(* IEC 61131-3 sources: Projecte/smart_office, 5 files *)

(* ---- control_cortines.st ---- *)
// 4. Màquina d'Estats
IF #HabilitarControl THEN
    CASE #Estat OF
        0: // Repòs
            #EnMoviment := FALSE;
            #VelocitatActual := 0.0;
            #RampaActiva := FALSE;
            #ComptePasos := 0;
            IF #sPosicioActual_Passos <> #PosicioDesitjadaPassos THEN
                #Estat := 10; // Passar a Preparar Moviment
            END_IF;

        10: // Preparar Moviment
            #EnMoviment := TRUE;
            #DireccioAssignada := (#PosicioDesitjadaPassos > #sPosicioActual_Passos) XOR NOT #DireccioPerObrir;
            #VelocitatActual := 10.0; // Velocitat inicial
            #RampaActiva := TRUE;
            #ComptePasos := 0;
            #Estat := 20; // Passar a Moviment
            #sTimerPols(IN := TRUE,
                        PT := #PT);
            #PasActual := FALSE;

        20: // Moviment
            #sTimerPols(IN := TRUE,
                        PT := #TempsPolsActual);

            IF #sTimerPols.Q THEN
                // Reiniciar el temporitzador per al següent pols

                // Generar pols i actualitzar direcció
                #PasActual := NOT #PasActual;
                #MotorPols := #PasActual;
                #MotorDireccio := #DireccioAssignada;

                // Actualitzar posició segons la direcció
                IF #DireccioAssignada = #DireccioPerObrir THEN
                    #sPosicioActual_Passos := #sPosicioActual_Passos + 1;
                ELSE
                    #sPosicioActual_Passos := #sPosicioActual_Passos - 1;
                END_IF;

                // Control de Rampa
                IF #RampaActiva THEN
                    #ComptePasos := #ComptePasos + 1;
                    IF #ComptePasos >= #PasosPerRampa THEN
                        #ComptePasos := 0;
                        IF #sPosicioActual_Passos < (#PosicioDesitjadaPassos + #CarreraTotal_Passos / 10) AND
                            #sPosicioActual_Passos > (#PosicioDesitjadaPassos - #CarreraTotal_Passos / 10) THEN
                            // Desaccelerar
                            #VelocitatActual := #VelocitatActual - #Desacceleracio;
                            IF #VelocitatActual <= 10.0 THEN
                                #VelocitatActual := 10.0;
                                #RampaActiva := FALSE; // Fi de la rampa
                            END_IF;
                        ELSE
                            // Accelerar
                            #VelocitatActual := #VelocitatActual + #Acceleracio;
                            IF #VelocitatActual >= 100.0 THEN
                                #VelocitatActual := 100.0;
                            END_IF;
                        END_IF;

                        IF #VelocitatActual <> 0.0 THEN
                            // Conversió més directa i segura
                            #TempsPolsActual := DINT_TO_TIME(REAL_TO_DINT(1000.0 / #VelocitatActual));
                        ELSE
                            #TempsPolsActual := #TempsPolsBase;
                        END_IF;
                    END_IF;
                END_IF;

                // Comprovar posició desitjada (SENSE SENSORS DE LÍMIT)
                IF #sPosicioActual_Passos = #PosicioDesitjadaPassos THEN
                    #Estat := 0; // Aturar moviment
                    #MotorPols := FALSE;
                    #EnMoviment := FALSE;
                    #RampaActiva := FALSE;
                    #ComptePasos := 0;
                END_IF;
            END_IF;

        ELSE // Error
            #Estat := 0;
            #MotorPols := FALSE;
            #EnMoviment := FALSE;
            #RampaActiva := FALSE;
            #ComptePasos := 0;
    END_CASE;
ELSE
    #MotorPols := FALSE;
    #EnMoviment := FALSE;
    #RampaActiva := FALSE;
    #ComptePasos := 0;
END_IF;                // Control de Rampa
                IF #RampaActiva THEN
                    #ComptePasos := #ComptePasos + 1;
                    IF #ComptePasos >= #PasosPerRampa THEN
                        #ComptePasos := 0;
                        IF #sPosicioActual_Passos < (#PosicioDesitjadaPassos + #CarreraTotal_Passos / 10) AND
                            #sPosicioActual_Passos > (#PosicioDesitjadaPassos - #CarreraTotal_Passos / 10) THEN
                            // Desaccelerar
                            #VelocitatActual := #VelocitatActual - #Desacceleracio;
                            IF #VelocitatActual <= 10.0 THEN
                                #VelocitatActual := 10.0;
                                #RampaActiva := FALSE; // Fi de la rampa
                            END_IF;
                        ELSE
                            // Accelerar
                            #VelocitatActual := #VelocitatActual + #Acceleracio;
                            IF #VelocitatActual >= 100.0 THEN
                                #VelocitatActual := 100.0;
                            END_IF;
                        END_IF;

                        IF #VelocitatActual <> 0.0 THEN
                            // Conversió més directa i segura
                            #TempsPolsActual := DINT_TO_TIME(REAL_TO_DINT(1000.0 / #VelocitatActual));
                        ELSE
                            #TempsPolsActual := #TempsPolsBase;
                        END_IF;
                    END_IF;
                END_IF;

                // Comprovar posició desitjada (SENSE SENSORS DE LÍMIT)
                IF #sPosicioActual_Passos = #PosicioDesitjadaPassos THEN
                    #Estat := 0; // Aturar moviment
                    #MotorPols := FALSE;
                    #EnMoviment := FALSE;
                    #RampaActiva := FALSE;
                    #ComptePasos := 0;
                END_IF;
            END_IF;

        ELSE // Error
            #Estat := 0;
            #MotorPols := FALSE;
            #EnMoviment := FALSE;
            #RampaActiva := FALSE;
            #ComptePasos := 0;
    END_CASE;

ELSE
    #MotorPols := FALSE;
    #EnMoviment := FALSE;
    #RampaActiva := FALSE;
    #ComptePasos := 0;
END_IF;

(* ---- control_temperatura.st ---- *)
// BLOC 1: INICIALITZACIÓ I DEFINICIÓ DE VARIABLES
VAR_INPUT
    SetPointNodeRED : Real;  // Setpoint rebut de Node-RED
    sensor_temp_jefe : Int;  // Entrada del sensor de Factory IO (%IW40)
    temperatura_DB : "temperatura_cap_DB";  // Referència al DB de temperatura
END_VAR

VAR_OUTPUT
    TemperaturaNodeRED : Real;  // Temperatura en graus per Node-RED
END_VAR

STATIC
    // Constants del sistema
    TEMP_MIN : Real := 0.0;           // Temperatura mínima permesa (canviat de 15.0)
    TEMP_MAX : Real := 50.0;          // Temperatura màxima permesa (canviat de 30.0)
    ZONA_MORTA : Real := 0.3;         // Marge de zona morta pel control
    HISTERESI : Real := 1.2;          // Factor d'histèresi
    TEMPS_MINIM_CANVI : Time := T#180S; // Temps mínim entre canvis de mode
    TAXA_ESCALFAMENT : Real := 0.1;    // Taxa d'escalfament simulada
    TAXA_REFREDAMENT : Real := 0.05;   // Taxa de refredament simulada

    // Variables de control i estat
    PrimeraExecucio : Bool := TRUE;   // Flag de primera execució
    EstemEnZonaMorta : Bool;          // Control d'histèresi
    ControlActiu : Bool;              // Estat del sistema
    ModeFred : Bool;                  // Mode refrigeració actiu
    ModeCalent : Bool;                // Mode calefacció actiu
    ModeActual : String;              // Mode actual en text

    // Variables de temperatura i sensors
    TemperaturaSimulada : Real;       // Temperatura simulada del sistema
    UltimaTemperaturaReal : Real;     // Última lectura vàlida
    TemperaturaReal : Real;           // Temperatura actual
    TemperaturaEscalada : Real;       // Temperatura processada
    ValorSensor : Real;               // Valor raw del sensor
    Valor_Raw_Sensor : Int;           // Valor enter del sensor

    // Variables de temps i simulació
    TempsActual : Time;               // Temps actual
    TempsAnterior : Time;             // Temps anterior
    DeltaTemps : Real;                // Interval de temps
    ProporcioSimulada : Real;         // Proporció per simulació
    ValorSensorSimulat : Int;         // Valor simulat

    // Variables de sortida i control
    SortidaPID : Real;                // Sortida del controlador PID
    SortidaEscalada : Real;           // Sortida escalada (0-100%)

    // Variables HMI/Monitorització
    HMI_TemperaturaActual : Real;     // Temperatura actual per HMI
    HMI_SetPoint : Real;              // SetPoint actual per HMI
    HMI_ModeActual : String;          // Mode de funcionament per HMI
    HMI_PercentatgeSortida : Real;    // Percentatge sortida per HMI

{REGION 'Declaració de variables PID'}
VAR_INPUT
    EN : Bool;              // Habilitació del PID
    Setpoint : Real;        // Valor desitjat de temperatura
    Input : Real;           // Valor actual de temperatura
END_VAR

VAR_OUTPUT
    Output : Real;          // Sortida del controlador PID
END_VAR

// 1. PROCESSAMENT DEL SENSOR DE TEMPERATURA
// Inicialització de variables de simulació
IF #PrimeraExecucio THEN
    #PrimeraExecucio := FALSE;
    #TemperaturaSimulada := #TEMP_MIN;
    #UltimaTemperaturaReal := #TEMP_MIN;
    #TemperaturaEscalada := #TEMP_MIN;
    #TempsAnterior := T#0MS;
END_IF;

// 2. CONTROL PRINCIPAL ON/OFF
IF NOT #ClimaOn THEN
    // Sistema desactivat - Reset de variables
    #ControlActiu := FALSE;
    #SortidaPID := 0.0;
    #SortidaEscalada := 0.0;
    #ModeFred := FALSE;
    #ModeCalent := FALSE;
    #ModeActual := 'OFF';
    // Mantenim la última temperatura quan està apagat
    #TemperaturaEscalada := #TemperaturaSimulada;
ELSE
    #ControlActiu := TRUE;
END_IF;

// 3. ACTUALITZACIÓ DEL TEMPS I SIMULACIÓ
// Actualitzar temps per la simulació utilitzant TON
#TimerSimulacio(IN := TRUE,
                PT := T#1S);  // Actualitzem cada segon

IF #TimerSimulacio.Q THEN
    #TempsActual := #TimerSimulacio.ET;

    // Calcular delta de temps (en segons)
    IF #TempsAnterior = T#0MS THEN
        #DeltaTemps := 0.1;  // Valor inicial per evitar pics
    ELSE
        #DeltaTemps := DINT_TO_REAL(TIME_TO_DINT(#TempsActual - #TempsAnterior)) / 1000.0;
    END_IF;

    #TempsAnterior := #TempsActual;
    #TimerSimulacio(IN := FALSE,
                    PT := T#1S);  // Reiniciar el timer
END_IF;

// Processar valor del sensor abans de la simulació
#ValorSensor := INT_TO_REAL(#sensor_temp_jefe);
#Valor_Raw_Sensor := #sensor_temp_jefe;

// Normalització i escalat del sensor actual
#Proporcio := #ValorSensor / 27648.0;
#TemperaturaReal := #Proporcio * (#TEMP_MAX - #TEMP_MIN) + #TEMP_MIN;
#TemperaturaEscalada := #TemperaturaReal;  // Utilitzem la temperatura real en lloc de la simulada

// Assignar al DB de temperatura utilitzant la referència
#temperatura_DB.TemperaturaEscalada := #TemperaturaEscalada;

// Validació del SetPoint
IF #SetPointNodeRED < #TEMP_MIN THEN
    #SetPointNodeRED := #TEMP_MIN;
ELSIF #SetPointNodeRED > #TEMP_MAX THEN
    #SetPointNodeRED := #TEMP_MAX;
END_IF;

// Debug dels valors - Actualitzem sempre
#proporcio_debug := #Proporcio;
#temp_real_debug := #TemperaturaReal;
#setpoint_debug := #SetPointNodeRED;
#temp_entrada_pid := #TemperaturaEscalada;
#setpoint_entrada_pid := #SetPointNodeRED;

// Simulació del comportament tèrmic sempre activa
IF #ControlActiu THEN
    IF #ModeFred THEN
        // Mode refrigeració - La sortida del PID refreda
        #TemperaturaSimulada := #TemperaturaSimulada - (#SortidaEscalada * #TAXA_ESCALFAMENT * #DeltaTemps);
    ELSE
        // Mode calefacció - La sortida del PID escalfa
        #TemperaturaSimulada := #TemperaturaSimulada + (#SortidaEscalada * #TAXA_ESCALFAMENT * #DeltaTemps);
    END_IF;

    // Simular pèrdua natural de temperatura
    IF #TemperaturaSimulada > #TEMP_MIN THEN
        #TemperaturaSimulada := #TemperaturaSimulada - (#TAXA_REFREDAMENT * #DeltaTemps);
    END_IF;

    // Limitar la temperatura simulada
    IF #TemperaturaSimulada < #TEMP_MIN THEN
        #TemperaturaSimulada := #TEMP_MIN;
    ELSIF #TemperaturaSimulada > #TEMP_MAX THEN
        #TemperaturaSimulada := #TEMP_MAX;
    END_IF;

    // Actualitzar temperatura escalada amb la simulada
    #TemperaturaEscalada := #TemperaturaSimulada;

    // Convertir temperatura simulada a format sensor (0-27648)
    #ProporcioSimulada := (#TemperaturaSimulada - #TEMP_MIN) / (#TEMP_MAX - #TEMP_MIN);
    #ValorSensorSimulat := REAL_TO_INT(#ProporcioSimulada * 27648.0);

    // Assignar al tag del sensor
    "sensor_temp_jefe" := #ValorSensorSimulat;
END_IF;

// Debug dels valors - Actualitzem sempre
#proporcio_debug := #ProporcioSimulada;
#temp_real_debug := #TemperaturaSimulada;
#setpoint_debug := #SetPointNodeRED;
#temp_entrada_pid := #TemperaturaEscalada;
#setpoint_entrada_pid := #SetPointNodeRED;

// 3. GESTIÓ DE MODES AMB TEMPORITZACIÓ
IF #ControlActiu THEN
    // Control de temps mínim entre canvis
    #TimerCanviMode(IN := #BotoFred OR #BotoCalent,
                    PT := #TEMPS_MINIM_CANVI);

    // Canvi de mode amb temporització
    IF #TimerCanviMode.Q THEN
        IF #BotoFred AND NOT #BotoCalent AND NOT #ModeFred THEN
            // Activació mode fred
            #ModeFred := TRUE;
            #ModeCalent := FALSE;
            #ModeActual := 'Fred';
        ELSIF #BotoCalent AND NOT #BotoFred AND NOT #ModeCalent THEN
            // Activació mode calent
            #ModeFred := FALSE;
            #ModeCalent := TRUE;
            #ModeActual := 'Calent';
        END_IF;
    END_IF;

    // 4. CONTROL PID I SORTIDA
    IF #ClimaOn THEN
        // Configuració del PID
        "Control_temperatura_oficina_cap"(
            EN := #ClimaOn,
            Setpoint := #SetPointNodeRED,
            Input := #TemperaturaEscalada
        );

        // Execució del PID si estem fora de la zona morta
        IF NOT #EstemEnZonaMorta THEN
            #SortidaPID := "Control_temperatura_oficina_cap".Output;
            // Gestió mode fred
            IF #ModeFred THEN
                #SortidaPID := -#SortidaPID;
            END_IF;

            // Limitació de la sortida amb més granularitat
            IF #SortidaPID < 0.0 THEN
                #SortidaEscalada := 0.0;
            ELSIF #SortidaPID > 100.0 THEN
                #SortidaEscalada := 100.0;
            ELSE
                #SortidaEscalada := #SortidaPID;
            END_IF;
        END_IF;
    ELSE
        "Control_temperatura_oficina_cap"(EN := FALSE);
    END_IF;
END_IF;

// BLOC 5: PROCESSAMENT DE SORTIDES
// Convertir temperatura simulada a format sensor
#ProporcioSimulada := (#TemperaturaSimulada - #TEMP_MIN) / (#TEMP_MAX - #TEMP_MIN);
#ValorSensorSimulat := REAL_TO_INT(#ProporcioSimulada * 27648.0);

// Assignar al tag del sensor (simulació)
"sensor_temp_jefe" := #ValorSensorSimulat;

// Actualitzar sortides físiques
#refredament := #ControlActiu AND #ModeFred AND (#SortidaEscalada > 10.0);
#calefaccio := #ControlActiu AND #ModeCalent AND (#SortidaEscalada > 10.0);

// BLOC 6: DIAGNÒSTIC I MONITORITZACIÓ
// Variables per monitorització
#HMI_TemperaturaActual := #TemperaturaSimulada;
#HMI_SetPoint := #SetPointNodeRED;
#HMI_ModeActual := #ModeActual;
#HMI_PercentatgeSortida := #SortidaEscalada;

// Actualitzar temperatura per Node-RED
#Temperatura := #TemperaturaEscalada;

(* ---- control_temperatura_final.st ---- *)
// BLOC 1: INICIALITZACIÓ I DEFINICIÓ DE VARIABLES
VAR_INPUT
    ClimaOn : Bool;         // Interruptor principal del sistema (0.0)
    BotoFred : Bool;        // Botó per activar mode refrigeració (des de Node-RED)
    BotoCalent : Bool;      // Botó per activar mode calefacció (des de Node-RED)
    SetPointNodeRED : Real; // Punt de consigna rebut de Node-RED (2.0)
    sensor_temp_jefe : Int; // Entrada del sensor de Factory IO (%IW40)
END_VAR

VAR_OUTPUT
    refredament : Bool;          // Sortida de refrigeració (276.0)
    calefaccio : Bool;          // Sortida de calefacció (276.1)
    HMI_TemperaturaActual : Real; // Temperatura actual per HMI (278.0)
    HMI_SetPoint : Real;         // Punt de consigna per HMI (282.0)
    HMI_ModeActual : String;     // Mode actual per HMI (286.0)
    HMI_PercentatgeSortida : Real; // Percentatge sortida per HMI (542.0)
    TemperaturaNodeRED : Real;   // Temperatura per Node-RED
END_VAR

STATIC
    // Constants del sistema
    TEMP_MIN : Real := 0.0;            // Temperatura mínima (680.0)
    TEMP_MAX : Real := 50.0;           // Temperatura màxima (684.0)
    ZONA_MORTA : Real := 0.3;          // Marge de zona morta (572.0)
    HISTERESI : Real := 1.2;           // Factor d'histèresi (688.0)
    TEMPS_MINIM_CANVI : Time := T#180S; // Temps mínim entre canvis (568.0)

    // Variables de control i estat
    ControlActiu : Bool;               // Estat del sistema (14.0)
    ModeFred : Bool := FALSE;          // Mode refrigeració actiu (546.0)
    ModeCalent : Bool := FALSE;        // Mode calefacció actiu (546.1)
    ModeActual : String;               // Mode actual (16.0)
    EstemEnZonaMorta : Bool;           // Control d'histèresi (600.0)

    // Variables de temperatura i sensors
    TemperaturaReal : Real;            // Temperatura actual (606.0)
    TemperaturaEscalada : Real;        // Temperatura processada (6.0)
    ValorSensor : Real;                // Valor del sensor (610.0)
    Proporcio : Real;                  // Proporció escalada (548.0)

    // Variables de sortida i control
    SortidaPID : Real;                 // Sortida del controlador PID (10.0)
    SortidaEscalada : Real;            // Sortida escalada 0-100% (272.0)

    // Timer per canvi de mode
    TimerCanviMode : TON_TIME;         // Timer pel canvi de mode (552.0)
END_STATIC

BEGIN
// BLOC 2: PROCESSAMENT DEL SENSOR
// Lectura i processament del sensor
#ValorSensor := INT_TO_REAL(#sensor_temp_jefe);  // Llegim el valor del potenciòmetre
#Proporcio := #ValorSensor / 27648.0;            // Normalitzem a 0-1
#TemperaturaReal := #Proporcio * (#TEMP_MAX - #TEMP_MIN) + #TEMP_MIN;  // Escalem a 0-50°C
#TemperaturaEscalada := #TemperaturaReal;

// BLOC 3: CONTROL PRINCIPAL
IF NOT #ClimaOn THEN
    // Sistema desactivat - Reset de variables
    #ControlActiu := FALSE;
    #SortidaPID := 0.0;
    #SortidaEscalada := 0.0;
    #ModeFred := FALSE;
    #ModeCalent := FALSE;
    #ModeActual := 'Aturat';
ELSE
    #ControlActiu := TRUE;
END_IF;

// BLOC 4: GESTIÓ DE MODES
IF #ControlActiu THEN
    // Control de temps mínim entre canvis
    #TimerCanviMode(IN := (#BotoFred AND NOT #ModeFred) OR (#BotoCalent AND NOT #ModeCalent),
                    PT := #TEMPS_MINIM_CANVI);

    // Actualització de modes amb temporització
    IF #TimerCanviMode.Q THEN
        #ModeFred := #BotoFred AND NOT #BotoCalent;
        #ModeCalent := #BotoCalent AND NOT #BotoFred;

        IF #ModeFred THEN
            #ModeActual := 'Fred';
        ELSIF #ModeCalent THEN
            #ModeActual := 'Calent';
        ELSE
            #ModeActual := 'Aturat';
        END_IF;
    END_IF;

    // BLOC 5: CONTROL PID
    IF #ClimaOn THEN
        // PID Mode Fred
        "Control_temperatura_fred"(
            EN := #ControlActiu AND #ModeFred,  // Cambiado de BotoFred a ModeFred
            ManualEnable := FALSE,
            Reset := FALSE,
            Setpoint := #SetPointNodeRED,
            Input := #TemperaturaEscalada,
            ManualValue := 0.0
        );

        // PID Mode Calent
        "Control_temperatura_calent"(
            EN := #ControlActiu AND #ModeCalent,  // Cambiado de BotoCalent a ModeCalent
            ManualEnable := FALSE,
            Reset := FALSE,
            Setpoint := #SetPointNodeRED,
            Input := #TemperaturaEscalada,
            ManualValue := 0.0
        );

        // Actualitzar zona morta
        #EstemEnZonaMorta := ABS(#SetPointNodeRED - #TemperaturaEscalada) < #ZONA_MORTA;

        // Selecció de la sortida segons el mode actiu
        IF #ModeFred AND NOT #EstemEnZonaMorta THEN  // Cambiado de BotoFred a ModeFred
            #SortidaPID := "Control_temperatura_fred".Output;
        ELSIF #ModeCalent AND NOT #EstemEnZonaMorta THEN  // Cambiado de BotoCalent a ModeCalent
            #SortidaPID := "Control_temperatura_calent".Output;
        END_IF;

        // Limitació de la sortida (comuna per ambdós modes)
        IF #SortidaPID < 0.0 THEN
            #SortidaEscalada := 0.0;
        ELSIF #SortidaPID > 100.0 THEN
            #SortidaEscalada := 100.0;
        ELSE
            #SortidaEscalada := #SortidaPID;
        END_IF;
    ELSE
        // Desactivem ambdós PIDs i els posem en mode manual
        "Control_temperatura_fred"(
            EN := FALSE,
            ManualEnable := TRUE,
            Reset := TRUE,
            Setpoint := 0.0,
            Input := 0.0,
            ManualValue := 0.0
        );

        "Control_temperatura_calent"(
            EN := FALSE,
            ManualEnable := TRUE,
            Reset := TRUE,
            Setpoint := 0.0,
            Input := 0.0,
            ManualValue := 0.0
        );
    END_IF;
END_IF;

// BLOC 6: ACTUALITZACIÓ DE SORTIDES
#refredament := #ControlActiu AND #ModeFred;  // En simulació, activem directament amb el mode
#calefaccio := #ControlActiu AND #ModeCalent;  // En simulació, activem directament amb el mode

// BLOC 7: ACTUALITZACIÓ DE VARIABLES HMI
#HMI_TemperaturaActual := #TemperaturaReal;
#HMI_SetPoint := #SetPointNodeRED;
#HMI_ModeActual := #ModeActual;
#HMI_PercentatgeSortida := #SortidaEscalada;

// Actualització Node-RED
#TemperaturaNodeRED := #TemperaturaReal;

END_PROGRAM

(* ---- control_temperatura_net.st ---- *)
// BLOC 1: INICIALITZACIÓ I DEFINICIÓ DE VARIABLES
VAR_INPUT
    ClimaOn : Bool;         // Interruptor principal del sistema (0.0)
    BotoFred : Bool;        // Botó per activar mode refrigeració (des de Node-RED)
    BotoCalent : Bool;      // Botó per activar mode calefacció (des de Node-RED)
    SetPointNodeRED : Real; // Punt de consigna rebut de Node-RED (2.0)
    sensor_temp_jefe : Int; // Entrada del sensor de Factory IO (%IW40)
END_VAR

VAR_OUTPUT
    refredament : Bool;          // Sortida de refrigeració (276.0)
    calefaccio : Bool;          // Sortida de calefacció (276.1)
    HMI_TemperaturaActual : Real; // Temperatura actual per HMI (278.0)
    HMI_SetPoint : Real;         // Punt de consigna per HMI (282.0)
    HMI_ModeActual : String;     // Mode actual per HMI (286.0)
    HMI_PercentatgeSortida : Real; // Percentatge sortida per HMI (542.0)
    TemperaturaNodeRED : Real;   // Temperatura per Node-RED
END_VAR

// No necessitem declarar el DB ja que utilitzem les variables de sortida

STATIC
    // Constants del sistema
    TEMP_MIN : Real := 0.0;            // Temperatura mínima (680.0)
    TEMP_MAX : Real := 50.0;           // Temperatura màxima (684.0)
    ZONA_MORTA : Real := 0.3;          // Marge de zona morta (572.0)
    HISTERESI : Real := 1.2;           // Factor d'histèresi (688.0)
    TEMPS_MINIM_CANVI : Time := T#180S; // Temps mínim entre canvis (568.0)

    // Variables de control i estat
    ControlActiu : Bool;               // Estat del sistema (14.0)
    ModeFred : Bool := FALSE;          // Mode refrigeració actiu (546.0)
    ModeCalent : Bool := FALSE;        // Mode calefacció actiu (546.1)
    ModeActual : String;               // Mode actual (16.0)
    EstemEnZonaMorta : Bool;           // Control d'histèresi (600.0)

    // Variables de temperatura i sensors
    TemperaturaReal : Real;            // Temperatura actual (606.0)
    TemperaturaEscalada : Real;        // Temperatura processada (6.0)
    ValorSensor : Real;                // Valor del sensor (610.0)
    Proporcio : Real;                  // Proporció escalada (548.0)

    // Variables de sortida i control
    SortidaPID : Real;                 // Sortida del controlador PID (10.0)
    SortidaEscalada : Real;            // Sortida escalada 0-100% (272.0)

    // Timer per canvi de mode
    TimerCanviMode : TON_TIME;         // Timer pel canvi de mode (552.0)
END_STATIC

BEGIN
// BLOC 2: PROCESSAMENT DEL SENSOR
// Lectura i processament del sensor
#ValorSensor := INT_TO_REAL(#sensor_temp_jefe);  // Llegim el valor del potenciòmetre
#Proporcio := #ValorSensor / 27648.0;            // Normalitzem a 0-1
#TemperaturaReal := #Proporcio * (#TEMP_MAX - #TEMP_MIN) + #TEMP_MIN;  // Escalem a 0-50°C
#TemperaturaEscalada := #TemperaturaReal;

// BLOC 3: CONTROL PRINCIPAL
IF NOT #ClimaOn THEN
    // Sistema desactivat - Reset de variables
    #ControlActiu := FALSE;
    #SortidaPID := 0.0;
    #SortidaEscalada := 0.0;
    #ModeFred := FALSE;
    #ModeCalent := FALSE;
    #ModeActual := 'Aturat';
ELSE
    #ControlActiu := TRUE;
END_IF;

// BLOC 4: GESTIÓ DE MODES
IF #ControlActiu THEN
    // Control de temps mínim entre canvis
    #TimerCanviMode(IN := #ModeNodeRED <> #ModeActual,
                    PT := #TEMPS_MINIM_CANVI);

    // Canvi de mode amb temporització
    IF #TimerCanviMode.Q THEN
        CASE #ModeNodeRED OF
            'Fred':
                #ModeFred := TRUE;
                #ModeCalent := FALSE;
                #ModeActual := 'Fred';
            'Calent':
                #ModeFred := FALSE;
                #ModeCalent := TRUE;
                #ModeActual := 'Calent';
        END_CASE;
    END_IF;    // BLOC 5: CONTROL PID
    IF #ClimaOn THEN
        // PID Mode Fred
        "Control_temperatura_fred"(
            EN := #ControlActiu AND #BotoFred,    // Activem només quan està en mode fred
            Setpoint := #SetPointNodeRED,
            Input := #TemperaturaEscalada
        );

        // PID Mode Calent
        "Control_temperatura_oficina_cap"(
            EN := #ControlActiu AND #BotoCalent,  // Activem només quan està en mode calent
            Setpoint := #SetPointNodeRED,
            Input := #TemperaturaEscalada
        );

        // Selecció de la sortida segons el mode actiu
        IF #BotoFred AND NOT #EstemEnZonaMorta THEN
            #SortidaPID := "Control_temperatura_fred".Output;
        ELSIF #BotoCalent AND NOT #EstemEnZonaMorta THEN
            #SortidaPID := "Control_temperatura_oficina_cap".Output;
        END_IF;

        // Limitació de la sortida (comuna per ambdós modes)
        IF #SortidaPID < 0.0 THEN
            #SortidaEscalada := 0.0;
        ELSIF #SortidaPID > 100.0 THEN
            #SortidaEscalada := 100.0;
        ELSE
            #SortidaEscalada := #SortidaPID;
        END_IF;
    ELSE
        // Desactivem ambdós PIDs
        "Control_temperatura_fred"(EN := FALSE);
        "Control_temperatura_oficina_cap"(EN := FALSE);
    END_IF;
END_IF;

// BLOC 6: ACTUALITZACIÓ DE SORTIDES
#refredament := #ControlActiu AND #ModeFred AND (#SortidaEscalada > 10.0);
#calefaccio := #ControlActiu AND #ModeCalent AND (#SortidaEscalada > 10.0);

// BLOC 7: ACTUALITZACIÓ DE VARIABLES HMI
#HMI_TemperaturaActual := #TemperaturaReal;
#HMI_SetPoint := #SetPointNodeRED;
#HMI_ModeActual := #ModeActual;
#HMI_PercentatgeSortida := #SortidaEscalada;

// Actualització Node-RED
#TemperaturaNodeRED := #TemperaturaReal;

END_PROGRAM

(* ---- control_temperatura_nou.st ---- *)
// BLOC 1: INICIALITZACIÓ I DEFINICIÓ DE VARIABLES
VAR_INPUT
    SetPointNodeRED : Real;  // Punt de consigna rebut de Node-RED
    sensor_temp_jefe : Int;  // Entrada del sensor de Factory IO (%IW40)
    temperatura_cap_DB : "temperatura_cap_DB";  // Referència al DB
    BotoFred : Bool;         // Botó per activar mode refrigeració
    BotoCalent : Bool;       // Botó per activar mode calefacció
    ClimaOn : Bool;         // Interruptor principal del sistema
END_VAR

VAR_OUTPUT
    TemperaturaNodeRED : Real;  // Temperatura en graus per Node-RED
    refredament : Bool;         // Sortida de refrigeració
    calefaccio : Bool;         // Sortida de calefacció
END_VAR

STATIC
    // Constants del sistema
    TEMP_MIN : Real := 0.0;           // Temperatura mínima permesa
    TEMP_MAX : Real := 50.0;          // Temperatura màxima permesa
    ZONA_MORTA : Real := 0.3;         // Marge de zona morta pel control
    HISTERESI : Real := 1.2;          // Factor d'histèresi
    TEMPS_MINIM_CANVI : Time := T#180S; // Temps mínim entre canvis de mode

    // Variables de control i estat
    EstemEnZonaMorta : Bool;          // Control d'histèresi
    ControlActiu : Bool;              // Estat del sistema
    ModeFred : Bool := FALSE;         // Mode refrigeració actiu
    ModeCalent : Bool := FALSE;       // Mode calefacció actiu
    ModeActual : String;              // Mode actual en text

    // Variables de temperatura i sensors
    TemperaturaReal : Real;           // Temperatura actual
    TemperaturaEscalada : Real;       // Temperatura processada
    ValorSensor : Real;               // Valor del sensor
    Proporcio : Real;                 // Proporció escalada del sensor

    // Variables de sortida i control
    SortidaPID : Real;                // Sortida del controlador PID
    SortidaEscalada : Real;           // Sortida escalada (0-100%)

    // Variables HMI/Monitorització
    HMI_TemperaturaActual : Real;     // Temperatura actual per HMI
    HMI_SetPoint : Real;              // Punt de consigna actual per HMI
    HMI_ModeActual : String;          // Mode de funcionament per HMI
    HMI_PercentatgeSortida : Real;    // Percentatge sortida per HMI
END_VAR

BEGIN
// BLOC 2: PROCESSAMENT DEL SENSOR
// Lectura i processament del sensor
#ValorSensor := INT_TO_REAL("sensor_temp_jefe");  // Llegim el valor del potenciòmetre
#Proporcio := #ValorSensor / 27648.0;            // Normalitzem a 0-1
#TemperaturaReal := #Proporcio * (#TEMP_MAX - #TEMP_MIN) + #TEMP_MIN;  // Escalem a 0-50°C
#TemperaturaEscalada := #TemperaturaReal;

// BLOC 3: CONTROL PRINCIPAL
IF NOT #ClimaOn THEN
    // Sistema desactivat - Reset de variables
    #ControlActiu := FALSE;
    #SortidaPID := 0.0;
    #SortidaEscalada := 0.0;
    #ModeFred := FALSE;
    #ModeCalent := FALSE;
    #ModeActual := 'Aturat';
ELSE
    #ControlActiu := TRUE;
END_IF;

// BLOC 4: GESTIÓ DE MODES
IF #ControlActiu THEN
    // Control de temps mínim entre canvis
    #TimerCanviMode(IN := #BotoFred OR #BotoCalent,
                    PT := #TEMPS_MINIM_CANVI);

    // Canvi de mode amb temporització
    IF #TimerCanviMode.Q THEN
        IF #BotoFred AND NOT #BotoCalent THEN
            #ModeFred := TRUE;
            #ModeCalent := FALSE;
            #ModeActual := 'Fred';
        ELSIF #BotoCalent AND NOT #BotoFred THEN
            #ModeFred := FALSE;
            #ModeCalent := TRUE;
            #ModeActual := 'Calent';
        END_IF;
    END_IF;

    // BLOC 5: CONTROL PID
    IF #ClimaOn THEN
        "Control_temperatura_oficina_cap"(
            EN := #ControlActiu,
            Setpoint := #SetPointNodeRED,
            Input := #TemperaturaEscalada
        );

        IF NOT #EstemEnZonaMorta THEN
            #SortidaPID := "Control_temperatura_oficina_cap".Output;

            // Inversió de sortida per mode fred
            IF #ModeFred THEN
                #SortidaPID := -#SortidaPID;
            END_IF;

            // Limitació de la sortida
            IF #SortidaPID < 0.0 THEN
                #SortidaEscalada := 0.0;
            ELSIF #SortidaPID > 100.0 THEN
                #SortidaEscalada := 100.0;
            ELSE
                #SortidaEscalada := #SortidaPID;
            END_IF;
        END_IF;
    ELSE
        "Control_temperatura_oficina_cap"(EN := FALSE);
    END_IF;
END_IF;

// BLOC 6: ACTUALITZACIÓ DE SORTIDES
#refredament := #ControlActiu AND #ModeFred AND (#SortidaEscalada > 10.0);
#calefaccio := #ControlActiu AND #ModeCalent AND (#SortidaEscalada > 10.0);

// BLOC 7: ACTUALITZACIÓ DE VARIABLES HMI I DB
#HMI_TemperaturaActual := #TemperaturaReal;
#HMI_SetPoint := #SetPointNodeRED;
#HMI_ModeActual := #ModeActual;
#HMI_PercentatgeSortida := #SortidaEscalada;

// Actualitzacions DB
#temperatura_cap_DB.TemperaturaEscalada := #TemperaturaEscalada;
#temperatura_cap_DB.HMI_TemperaturaActual := #TemperaturaReal;
#temperatura_cap_DB.HMI_SetPoint := #SetPointNodeRED;

// Actualització Node-RED
#TemperaturaNodeRED := #TemperaturaReal;

END_PROGRAM
